(* IEC 61131-3 sources: AXOpen/src/data/ctrl/src, 20 files *)

(* ---- AxoDataCrudTask.st ---- *)
USING AXOpen.Core;

NAMESPACE AXOpen.Data

    ///<summary>
    /// Provides remote execution for CRUD operations.
    /// > [!NOTE]
    /// > This is an extension of <see cref="AxoTask"/>task see the documentatio for details about implementation in .NET.
    /// </summary>
    {#ix-set:AttributeName = "<#Data operation#>"}
    {S7.extern=ReadWrite}
    CLASS AxoDataCrudTask EXTENDS AxoRemoteTask IMPLEMENTS IAxoDataCrudTaskEntityExistState
        VAR PUBLIC
            ///<summary>
            /// Gets or sets the type of CRUD operation to be perfomed.
            /// </summary>
            CrudOperation : eCrudOperation;
            DataEntityIdentifier : STRING[254];
            _exist : BOOL;
        END_VAR

        VAR PRIVATE
            _LastCrudOperation : eCrudOperation;
            _LastDataEntityIdentifier : STRING[254];
        END_VAR
        ///<summary>
        /// Invokes this task.
        /// </summary>
        /// <param name="identifier">Data entity identifier</param>
        /// <param name="operation">Operation to perfom.</param>
        METHOD PUBLIC Invoke : IAxoTaskState
            VAR_INPUT
                identifier : STRING[254];
                operation : eCrudOperation;
            END_VAR

            // This may produce unwanted side effects if the task is invoked with different parameters while it is running.
            // It may prevent done state to be provided upstream to the caller.
            IF SUPER.IsDone() THEN
                IF (_LastDataEntityIdentifier   <> identifier OR
                    _LastCrudOperation          <> operation ) THEN
                    SUPER.Restore();
                END_IF;
            END_IF;

            IF SUPER.IsReady() THEN
                DataEntityIdentifier := identifier;
                CrudOperation := operation;
            END_IF;

            _LastDataEntityIdentifier   := DataEntityIdentifier;
            _LastCrudOperation          := CrudOperation;

            Invoke := SUPER.Invoke();
        END_METHOD

        METHOD PUBLIC Exist : BOOL
            Exist := _exist;
        END_METHOD

    END_CLASS

    TYPE
        eCrudOperation : (Create, Read, Update, Delete, CreateOrUpdate, EntityExist);
    END_TYPE
END_NAMESPACE

(* ---- AxoDataPersistentCurdTask.st ---- *)
USING AXOpen.Core;
NAMESPACE AXOpen.Data
    ///<summary>
    /// Provides remote execution for CRUD operations.
    /// > [!NOTE]
    /// > This is an extension of <see cref="AxoTask"/>task see the documentation for details about implementation in .NET.
    /// </summary>
    {#ix-set:AttributeName = "<#Data operation#>"}
    {S7.extern=ReadWrite}
    CLASS AxoDataPersistentCurdTask EXTENDS AxOpen.Core.AxoRemoteTask IMPLEMENTS  IAxoDataCrudTaskEntityExistState
        VAR PUBLIC
            ///<summary>
            /// Gets or sets the type of CRUD operation to be perfomed.
            /// </summary>
            CrudOperation : ePersistentOperation;
            DataEntityIdentifier : STRING[254];
            _exist : BOOL;
        END_VAR

        ///<summary>
        /// Invokes this task.
        /// </summary>
        /// <param name="identifier">Data entity identifier</param>
        /// <param name="operation">Operation to perfom.</param>
        METHOD PUBLIC Invoke : IAxoTaskState
            VAR_INPUT
                identifier : STRING[254];
                operation : ePersistentOperation;
            END_VAR
            CrudOperation := operation;
            DataEntityIdentifier := identifier;
            Invoke := SUPER.Invoke();
        END_METHOD

        METHOD PUBLIC Exist : BOOL
            Exist := _exist;
        END_METHOD

    END_CLASS

    TYPE
        ePersistentOperation : (Read, Update, EntityExist, UpdateAll, ReadAll);
    END_TYPE

END_NAMESPACE

(* ---- AxoDataEntityExistTask.st ---- *)
USING AXOpen.Core;

NAMESPACE AXOpen.Data
    ///<summary>
    /// Extends AxoRemoteTask for data operation within AxoData
    /// </summary>
    CLASS AxoDataEntityExistTask
        EXTENDS AxoDataExchangeTask
        IMPLEMENTS IAxoDataEntityExistTask
        VAR PUBLIC
            _exist : BOOL;
        END_VAR

        METHOD PUBLIC Exist : BOOL
            Exist := _exist;
        END_METHOD
    END_CLASS

    INTERFACE PUBLIC IAxoDataEntityExistTask EXTENDS IAxoTaskState
        METHOD Exist : BOOL END_METHOD
    END_INTERFACE

END_NAMESPACE

(* ---- AxoDataExchangeBase.st ---- *)
USING AXOpen.Core;

NAMESPACE AXOpen.Data
    ///<summary>
    /// Represents base class of data exchange.
    /// This class is used to provide abstract information about the type that can be used in rcc.
    /// </summary>
    INTERFACE PUBLIC AxoDataExchangeBase EXTENDS AXOpen.Core.IAxoObject
    END_INTERFACE
END_NAMESPACE

(* ---- IAxoDataCrudTaskEntityExistState.st ---- *)
NAMESPACE AXOpen.Data
    INTERFACE PUBLIC IAxoDataCrudTaskEntityExistState EXTENDS AXOpen.Core.IAxoTaskState
            METHOD Exist : BOOL END_METHOD
    END_INTERFACE
END_NAMESPACE

(* ---- IAxoDataEntity.st ---- *)
NAMESPACE AXOpen.Data
    INTERFACE IAxoDataEntity
        METHOD SetId
            VAR_INPUT
                Id : STRING[254];
            END_VAR
        END_METHOD
        METHOD GetId : STRING[254] END_METHOD

    END_INTERFACE
END_NAMESPACE

(* ---- IAxoDataExchange.st ---- *)
USING AXOpen.Core;

NAMESPACE AXOpen.Data
    ///<summary>
    /// Provides abastaction for data exchange.
    /// </summary>
    INTERFACE IAxoDataExchange
        METHOD Create : IAxoTaskState
            VAR_INPUT
                inIdentifier : STRING[254];
            END_VAR
        END_METHOD

        METHOD Read : IAxoTaskState
            VAR_INPUT
                inIdentifier : STRING[254];
            END_VAR
        END_METHOD

        METHOD Update : IAxoTaskState
            VAR_INPUT
                inIdentifier : STRING[254];
            END_VAR
        END_METHOD

        METHOD Delete : IAxoTaskState
            VAR_INPUT
                inIdentifier : STRING[254];
            END_VAR
        END_METHOD

        METHOD EntityExist : IAxoDataCrudTaskEntityExistState
            VAR_INPUT
                inIdentifier : STRING[254];
            END_VAR
        END_METHOD

        METHOD CreateOrUpdate : IAxoTaskState
            VAR_INPUT
                inIdentifier : STRING[254];
            END_VAR
        END_METHOD

        METHOD Restore
        END_METHOD

        METHOD Run
            VAR_INPUT
                inParent : IAxoObject;
            END_VAR
        END_METHOD
    END_INTERFACE
END_NAMESPACE

(* ---- IDataEntity.st ---- *)
NAMESPACE AXOpen.Data
    INTERFACE IDataEntity

    END_INTERFACE
END_NAMESPACE

(* ---- IDataExchange.st ---- *)
USING AXOpen.Core;

NAMESPACE ix.framework.data
    INTERFACE IDataExchange
        METHOD Create : IAxoTaskState
            VAR_INPUT
                Identifier : STRING[254];
            END_VAR
        END_METHOD

        METHOD Read : IAxoTaskState
            VAR_INPUT
                Identifier : STRING[254];
            END_VAR
        END_METHOD

        METHOD Update : IAxoTaskState
            VAR_INPUT
                Identifier : STRING[254];
            END_VAR
        END_METHOD

        METHOD Delete : IAxoTaskState
            VAR_INPUT
                Identifier : STRING[254];
            END_VAR
        END_METHOD

        METHOD Restore
        END_METHOD
    END_INTERFACE
END_NAMESPACE

(* ---- AxoDataCrudTaskEntityExistsSatisfied.st ---- *)
NAMESPACE AXOpen.Data

    ///<summary>
    /// Represents the satisfied state of a data CRUD task entity existence check.
    /// </summary>
    CLASS PUBLIC AxoDataCrudTaskEntityExistsSatisfied EXTENDS AXOpen.Core.AxoTaskStateSatisfied IMPLEMENTS IAxoDataCrudTaskEntityExistState
        VAR PRIVATE
            _exists : BOOL;
        END_VAR

        ///<summary>
        /// Returns true when the entity exists. Prior to calling this method you should call Satisfy.
        /// </summary>
        METHOD PUBLIC Exist : BOOL
            Exist := _exists;
            _exists := FALSE;
        END_METHOD

        ///<summary>
        /// Satisfies the task state by setting the existence status.
        /// </summary>
        METHOD PUBLIC Satisfy : IAxoDataCrudTaskEntityExistState
            VAR_INPUT
                inStatus : eAxoTaskState;
                inDoesExist : BOOL;
            END_VAR
            Status := inStatus;
            _exists := inDoesExist;
            Satisfy := THIS;
        END_METHOD
    END_CLASS
END_NAMESPACE

(* ---- AxoDataEntity.st ---- *)
USING AXOpen.Core;
NAMESPACE AXOpen.Data
    ///<summary>
    /// Base class for any exchangable data in <see cref="AxoDataExchange"/>.
    /// </summary>
    {S7.extern=ReadWrite}
    CLASS AxoDataEntity IMPLEMENTS IAxoDataEntity
        VAR PUBLIC
            ///<summary>
            /// Gets or sets data entity identifier.
            /// </summary>
            {#ix-attr:[RenderIgnore()]}
            DataEntityId : STRING[254];
        END_VAR

        METHOD PUBLIC SetId
            VAR_INPUT
                Id : STRING[254];
            END_VAR
            DataEntityId := Id;
        END_METHOD

        METHOD PUBLIC GetId : STRING[254]
            GetId := DataEntityId;
        END_METHOD
    END_CLASS
END_NAMESPACE

(* ---- AxoDataExchange.st ---- *)
USING AXOpen.Core;

NAMESPACE AXOpen.Data
    ///<summary>
    /// Provides base class for any data exchange with an arbitrary remote repository.
    /// </summary>
    {#ix-generic:<TOnline, TPlain>}
    {S7.extern=ReadWrite}
    CLASS AxoDataExchange EXTENDS AxoObject IMPLEMENTS IAxoDataExchange, AxoDataExchangeBase
        VAR PUBLIC
            Operation : AxoDataCrudTask;
        END_VAR

        ///<summary>
        /// Runs intialization and cyclical handling of this AxoDataExchange.
        /// </summary>
        /// <param name="parent">Parent of this object</param>
        METHOD PUBLIC OVERRIDE Run
            VAR_INPUT
                inParent : IAxoObject;
            END_VAR
            SUPER.Run(inParent);
            // Operation.Run(THIS);
            Operation.Execute(THIS);
        END_METHOD

        ///<summary>
        /// Creates new entry into the remote repository from data entity of this AxoDataExchange.
        /// </summary>
        /// <param name="identifier">Data identifier.</param>
        METHOD PUBLIC Create : IAxoTaskState
            VAR_INPUT
                identifier : STRING[254];
            END_VAR
            Create := Operation.Invoke(identifier, eCrudOperation#Create);
        END_METHOD

        ///<summary>
        /// Reads data from remote repository and copies them into data entity of this AxoDataExchange.
        /// </summary>
        /// <param name="identifier">Data identifier.</param>
        METHOD PUBLIC Read : IAxoTaskState
            VAR_INPUT
                identifier : STRING[254];
            END_VAR
            Read := Operation.Invoke(identifier, eCrudOperation#Read);
        END_METHOD

        ///<summary>
        /// Updates data in remote repository from data entiry of this AxoDataExchange.
        /// </summary>
        /// <param name="identifier">Data identifier.</param>
        METHOD PUBLIC Update : IAxoTaskState
            VAR_INPUT
                identifier : STRING[254];
            END_VAR
            Update := Operation.Invoke(identifier, eCrudOperation#Update);
        END_METHOD

        ///<summary>
        /// Deletes data entry with given ID from remote repository.
        /// </summary>
        /// <param name="identifier">Data identifier.</param>
        METHOD PUBLIC Delete : IAxoTaskState
            VAR_INPUT
                identifier : STRING[254];
            END_VAR
            Delete := Operation.Invoke(identifier, eCrudOperation#Delete);
        END_METHOD

        ///<summary>
        /// Check if data entry exists with given ID in remote repository.
        /// </summary>
        /// <param name="identifier">Data identifier.</param>
        METHOD PUBLIC EntityExist : IAxoDataCrudTaskEntityExistState
            VAR_INPUT
                identifier : STRING[254];
            END_VAR
            Operation.Invoke(identifier, eCrudOperation#EntityExist);
            EntityExist := Operation;
        END_METHOD

        ///<summary>
        /// Creates or Updates data in remote repository from data entiry of this AxoDataExchange.
        /// </summary>
        /// <param name="identifier">Data identifier.</param>
        METHOD PUBLIC CreateOrUpdate : IAxoTaskState
            VAR_INPUT
                identifier : STRING[254];
            END_VAR
            CreateOrUpdate := Operation.Invoke(identifier, eCrudOperation#CreateOrUpdate);
        END_METHOD

        ///<summary>
        /// Restores all tasks associated with this object.
        ///</summary>
        METHOD PUBLIC Restore
            Operation.Restore();
        END_METHOD
    END_CLASS
END_NAMESPACE

(* ---- AxoDataExchangeTask.st ---- *)
USING AXOpen.Core;

NAMESPACE AXOpen.Data
    ///<summary>
    /// Extends AxoRemoteTask for data operation within AxoData
    /// </summary>
    CLASS AxoDataExchangeTask
        EXTENDS AXOpen.Core.AxoRemoteTask
        VAR PUBLIC
            DataEntityIdentifier : STRING[254];
        END_VAR

        METHOD PUBLIC Invoke : IAxoTaskState
            VAR_INPUT
                identifier : STRING[254];
            END_VAR
            DataEntityIdentifier := identifier;
            Invoke := SUPER.Invoke();
        END_METHOD
    END_CLASS

END_NAMESPACE

(* ---- AxoDataFragmentExchange.st ---- *)
USING AXOpen.Core;
NAMESPACE AXOpen.Data
    ///<summary>
    /// Provides base class for any composite/fragmetes data exchange combining one or more AxoDataExchange object.
    /// </summary>
    {S7.extern=ReadWrite}
    CLASS PUBLIC AxoDataFragmentExchange EXTENDS AxoObject IMPLEMENTS IAxoDataExchange, AxoDataExchangeBase
        VAR PUBLIC
            Operation : AxoDataCrudTask;
        END_VAR

        ///<summary>
        /// Creates new entry into each associated remote repository from respective data entity.
        /// </summary>
        /// <param name="identifier">Data identifier.</param>
        METHOD PUBLIC Create : IAxoTaskState
            VAR_INPUT
                inIdentifier : STRING[254];
            END_VAR
            Create := Operation.Invoke(inIdentifier, eCrudOperation#Create);
        END_METHOD

        ///<summary>
        /// Reads data from each associated remote repository and copies it into respective data entities.
        /// </summary>
        /// <param name="identifier">Data identifier.</param>
        METHOD PUBLIC Read : IAxoTaskState
            VAR_INPUT
                inIdentifier : STRING[254];
            END_VAR
            Read := Operation.Invoke(inIdentifier, eCrudOperation#Read);
        END_METHOD

        ///<summary>
        /// Updates data in each associated remote repository from respective data entities.
        /// </summary>
        /// <param name="identifier">Data identifier.</param>
        METHOD PUBLIC Update : IAxoTaskState
            VAR_INPUT
                inIdentifier : STRING[254];
            END_VAR
            Update := Operation.Invoke(inIdentifier, eCrudOperation#Update);
        END_METHOD

        ///<summary>
        /// Deletes data entry from each associated remote repository with given ID.
        /// </summary>
        /// <param name="identifier">Data identifier.</param>
        METHOD PUBLIC Delete : IAxoTaskState
            VAR_INPUT
                inIdentifier : STRING[254];
            END_VAR
            Delete := Operation.Invoke(inIdentifier, eCrudOperation#Delete);
        END_METHOD

        ///<summary>
        /// Check if data entry exists in each associated remote repository with given ID.
        /// </summary>
        /// <param name="identifier">Data identifier.</param>
        METHOD PUBLIC EntityExist : IAxoDataCrudTaskEntityExistState
            VAR_INPUT
                inIdentifier : STRING[254];
            END_VAR
            Operation.Invoke(inIdentifier, eCrudOperation#EntityExist);
            EntityExist := Operation;
        END_METHOD

        ///<summary>
        /// Creates or Updates data entry from each associated remote repository with given ID.
        /// </summary>
        /// <param name="identifier">Data identifier.</param>
        METHOD PUBLIC CreateOrUpdate : IAxoTaskState
            VAR_INPUT
                inIdentifier : STRING[254];
            END_VAR
            CreateOrUpdate := Operation.Invoke(inIdentifier, eCrudOperation#CreateOrUpdate);
        END_METHOD

        METHOD PUBLIC Restore
            Operation.Restore();
        END_METHOD

        ///<summary>
        /// Runs intialization and cyclical handling of this AxoDataExchange.
        /// </summary>
        /// <param name="parent">Parent of this object</param>
        METHOD PUBLIC OVERRIDE Run
            VAR_INPUT
                inParent : IAxoObject;
            END_VAR
            SUPER.Run(inParent);
            // Operation.Run(THIS);
            Operation.Execute(THIS);
        END_METHOD

    END_CLASS
END_NAMESPACE

(* ---- AxoDataLocalExchange.st ---- *)
NAMESPACE AXOpen.Data
    USING AXOpen.Core;

    ///<summary>
    /// Base class for any exchangable data in <see cref="AxoDataExchange"/>.
    /// </summary>
    {S7.extern=ReadWrite}
    CLASS PUBLIC ABSTRACT AxoDataLocalExchange EXTENDS AxoObject IMPLEMENTS IAxoDataExchange
        VAR  PROTECTED
            operation : eCrudOperation;
            dataExchangeTask : AxoTask;
        END_VAR

        METHOD PUBLIC Run
            VAR_INPUT
                inParent : IAxoObject;
            END_VAR
            ;
        END_METHOD

        METHOD PUBLIC ABSTRACT Create : IAxoTaskState
            VAR_INPUT
                Identifier : STRING[254];
            END_VAR

        END_METHOD

        METHOD PUBLIC ABSTRACT Read : IAxoTaskState
            VAR_INPUT
                Identifier : STRING[254];
            END_VAR

        END_METHOD

        METHOD PUBLIC ABSTRACT Update : IAxoTaskState
            VAR_INPUT
                Identifier : STRING[254];
            END_VAR

        END_METHOD

        METHOD PUBLIC ABSTRACT Delete : IAxoTaskState
            VAR_INPUT
                Identifier : STRING[254];
            END_VAR

        END_METHOD

        METHOD PUBLIC ABSTRACT EntityExist : IAxoEntityExistTaskState
            VAR_INPUT
                Identifier : STRING[254];
            END_VAR

        END_METHOD

        METHOD PUBLIC ABSTRACT CreateOrUpdate : IAxoTaskState
            VAR_INPUT
                Identifier : STRING[254];
            END_VAR

        END_METHOD

        METHOD PUBLIC Restore
            ;
        END_METHOD
    END_CLASS
END_NAMESPACE

(* ---- AxoDataPersistentExchange.st ---- *)
USING AXOpen.Core;
NAMESPACE AXOpen.Data
    {S7.extern=ReadWrite}
    CLASS PUBLIC AxoDataPersistentExchange EXTENDS AXOpen.Core.AxoObject
        VAR PUBLIC
            Operation : AxoDataPersistentCurdTask;
        END_VAR

        VAR CONSTANT
            DEFAULT_ID : STRING := 'default';
        END_VAR

        VAR
            _IsFirstReadAllDone  : BOOL := FALSE;

            // concurrent invoke handling...
            LastCallerIdentity : ULINT;
            LastCycleCount : ULINT;
            LastOperation : ePersistentOperation;

        END_VAR

        VAR PRIVATE
            _context : IAxoContext;
        END_VAR

        ///<summary>
        /// This method determines if the current call is concurrent or not.
        ///  It takes an AXOpen.Core.IAxoObject as input and returns a BOOL.
        /// The logic involves checking the identity of the caller and comparing it with the last caller identity,
        /// along with the operation's readiness and cycle count checks.
        /// </summary>
        /// <param name="caller">IAxoObject for identifying the caller in the context of concurrent calls</param>
        METHOD PRIVATE IsNotConcurrentCall : BOOL
            VAR_INPUT
                caller : AXOpen.Core.IAxoObject;
            END_VAR
            VAR
                newCallerIdentity : ULINT;
                newCycleCount : ULINT;
                operationState : eAxoTaskState;
            END_VAR

            IsNotConcurrentCall := false;
            newCallerIdentity := caller.GetIdentity();
            newCycleCount := THIS.GetContext().OpenCycleCount();

            IF newCallerIdentity = ULINT#0 THEN // IF IDENTITY IS NOT SET DO NOT ALLOW CALL
                RETURN;
            END_IF;

            IF  newCallerIdentity = LastCallerIdentity THEN
                IsNotConcurrentCall := true;
                LastCycleCount := newCycleCount;
                RETURN;
            ELSE
                operationState := Operation.GetState();
                IF (operationState = eAxoTaskState#Ready) OR (operationState = eAxoTaskState#Done)  THEN
                    IF LastCycleCount > newCycleCount THEN // counter overflow
                        IsNotConcurrentCall := true;
                        LastCycleCount := newCycleCount;
                        LastCallerIdentity := newCallerIdentity;
                        Operation.Restore();

                    ELSIF  (LastCycleCount + ULINT#2) < newCycleCount THEN
                        IsNotConcurrentCall := true;
                        LastCycleCount := newCycleCount;
                        LastCallerIdentity := newCallerIdentity;
                        Operation.Restore();
                    END_IF;
                END_IF;
            END_IF;

        END_METHOD

        ///<summary>
        /// Runs intialization and cyclical handling of this AxoDataPersistentExchange.
        /// </summary>
        /// <param name="parent">Parent of this object</param>
        METHOD PUBLIC OVERRIDE Run
            VAR_INPUT
                inParent : IAxoObject;
            END_VAR

            IF inParent = NULL THEN
                RETURN;
            END_IF;

            IF _context = NULL THEN
                SUPER.Run(inParent);
                Operation.Run(THIS);
                _context := THIS.GetContext();
            END_IF;

            Operation.Execute(THIS);

            IF NOT _IsFirstReadAllDone THEN
                IF Operation.IsInitialized AND (Operation.Identity <> ULINT#0) THEN // MUST BE INITIALIZED AND WITH IDENTITY
                    IF Operation.IsReady() THEN // read all after startup
                        Operation.Invoke('', ePersistentOperation#ReadAll);
                        LastOperation := ePersistentOperation#ReadAll;

                    ELSIF Operation.IsDone() AND (LastOperation = ePersistentOperation#ReadAll) THEN
                         _IsFirstReadAllDone := TRUE;
                    END_IF;
                END_IF;
            END_IF;
        END_METHOD

        ///<summary>
        /// Executes the restore Operation for the AxoDataPersistentExchange component.
        /// </summary>
        METHOD PUBLIC Restore
            Operation.Restore();
        END_METHOD

        /// <summary>
        /// Return last result of EntitiyExist Operation. True = Record Exist.
        /// </summary>
        METHOD PUBLIC EntityExistResult : BOOL
            EntityExistResult := Operation._exist;
        END_METHOD

        /// <summary>
        /// This method attempts to invoke a read operation.
        /// It checks if the call is concurrent and, if not,
        /// invokes the read operation on the Operation object.
        /// </summary>
        /// <param name="caller">IAxoObject for identifying the caller in the context of concurrent calls</param>
        /// <param name="identifier">The data identifier for the persistent group.</param>
        METHOD PUBLIC InvokeRead : BOOL
            VAR_INPUT
                caller : IAxoObject;
                identifier : STRING[254];
            END_VAR

            InvokeRead := false;
            IF _IsFirstReadAllDone THEN
                IF THIS.IsNotConcurrentCall(caller) THEN
                    InvokeRead := Operation.Invoke(identifier, ePersistentOperation#Read).IsBusy();
                    LastOperation := ePersistentOperation#Read;
                END_IF;
            END_IF;
        END_METHOD

        /// <summary>
        /// This method attempts to invoke a read operation.
        /// It checks if the call is concurrent and, if not,
        /// invokes the read operation on the Operation object.
        /// </summary>
        /// <param name="caller">IAxoObject for identifying the caller in the context of concurrent calls</param>
        METHOD PUBLIC InvokeReadDefault : BOOL
            VAR_INPUT
                caller : IAxoObject;
            END_VAR
            InvokeReadDefault := false;

            IF _IsFirstReadAllDone THEN
                IF THIS.IsNotConcurrentCall(caller) THEN
                    InvokeReadDefault := Operation.Invoke(DEFAULT_ID, ePersistentOperation#Read).IsBusy();
                    LastOperation := ePersistentOperation#Read;
                END_IF;
            END_IF;
        END_METHOD

        /// <summary>
        /// This method attempts to invoke a update operation.
        /// It checks if the call is concurrent and, if not,
        /// invokes the update operation on the Operation object.
        /// </summary>
        /// <param name="caller">IAxoObject for identifying the caller in the context of concurrent calls</param>
        /// <param name="identifier">The data identifier for the persistent group.</param>
        METHOD PUBLIC InvokeUpdate : BOOL
            VAR_INPUT
                Caller : IAxoObject;
                identifier : STRING[254];
            END_VAR
            InvokeUpdate := false;

            IF _IsFirstReadAllDone THEN
                IF THIS.IsNotConcurrentCall(Caller) THEN
                    InvokeUpdate := Operation.Invoke(identifier, ePersistentOperation#Update).IsBusy();
                    LastOperation := ePersistentOperation#Update;
                END_IF;
            END_IF;
        END_METHOD

        /// <summary>
        /// This method attempts to invoke a update operation.
        /// It checks if the call is concurrent and, if not,
        /// invokes the update operation on the Operation object.
        /// </summary>
        /// <param name="caller">IAxoObject for identifying the caller in the context of concurrent calls</param>
        METHOD PUBLIC InvokeUpdateDefault : BOOL
            VAR_INPUT
                Caller : IAxoObject;
            END_VAR
            InvokeUpdateDefault := false;

            IF _IsFirstReadAllDone THEN
                IF THIS.IsNotConcurrentCall(Caller) THEN
                    InvokeUpdateDefault := Operation.Invoke(DEFAULT_ID, ePersistentOperation#Update).IsBusy();
                    LastOperation := ePersistentOperation#Update;
                END_IF;
            END_IF;
        END_METHOD

        /// <summary>
        /// This method attempts to invoke a updateAll operation.
        /// It checks if the call is concurrent and, if not,
        /// invokes the update operation on the Operation object.
        /// </summary>
        /// <param name="caller">IAxoObject for identifying the caller in the context of concurrent calls</param>
        /// <param name="identifier">The data identifier for the persistent group.</param>
        METHOD PUBLIC InvokeUpdateAll : BOOL
            VAR_INPUT
                Caller : IAxoObject;
            END_VAR
            InvokeUpdateAll := false;

            IF _IsFirstReadAllDone THEN
                IF THIS.IsNotConcurrentCall(Caller) THEN
                    InvokeUpdateAll := Operation.Invoke('', ePersistentOperation#UpdateAll).IsBusy();
                    LastOperation := ePersistentOperation#UpdateAll;
                END_IF;
            END_IF;
        END_METHOD

        /// <summary>
        /// This method attempts to invoke a readAll operation.
        /// It checks if the call is concurrent and, if not,
        /// invokes the readAll operation on the Operation object.
        /// </summary>
        /// <param name="caller">IAxoObject for identifying the caller in the context of concurrent calls</param>
        /// <param name="identifier">The data identifier for the persistent group.</param>
        METHOD PUBLIC InvokeReadAll : BOOL
            VAR_INPUT
                Caller : IAxoObject;
            END_VAR
            InvokeReadAll := false;

            IF _IsFirstReadAllDone THEN
                IF THIS.IsNotConcurrentCall(Caller) THEN
                    InvokeReadAll := Operation.Invoke('', ePersistentOperation#ReadAll).IsBusy();
                    LastOperation := ePersistentOperation#ReadAll;
                END_IF;
            END_IF;
        END_METHOD

        /// <summary>
        /// This method attempts to invoke a update operation.
        /// It checks if the call is concurrent and, if not,
        /// invokes the update operation on the Operation object.
        /// </summary>
        /// <param name="caller">IAxoObject for identifying the caller in the context of concurrent calls</param>
        /// <param name="identifier">The data identifier for the persistent group.</param>
        METHOD PUBLIC InvokeEntityExist : BOOL
            VAR_INPUT
                Caller : IAxoObject;
                identifier : STRING[254];
            END_VAR

            InvokeEntityExist := false;
            IF _IsFirstReadAllDone THEN
                IF THIS.IsNotConcurrentCall(Caller) THEN
                    InvokeEntityExist := Operation.Invoke(identifier, ePersistentOperation#EntityExist).IsBusy();
                    LastOperation := ePersistentOperation#EntityExist;
                END_IF;
            END_IF;
        END_METHOD

        /// <summary>
        /// Determines whether a read operation has been completed.
        /// </summary>
        /// <param name="caller">The object representing the caller of the method, used to check for concurrent calls.</param>
        /// <returns>Boolean indicating whether the read operation was completed.</returns>
        METHOD PUBLIC IsReadDone : BOOL
            VAR_INPUT
                caller : IAxoObject;
            END_VAR
            IsReadDone := false;

            IF _IsFirstReadAllDone THEN
                IF THIS.IsNotConcurrentCall(caller) THEN
                    IF LastOperation = ePersistentOperation#Read THEN
                        IsReadDone := Operation.IsDone();
                    END_IF;
                END_IF;
            END_IF;
        END_METHOD

        /// <summary>
        /// Determines whether a update operation has been completed.
        /// </summary>
        /// <param name="caller">The object representing the caller of the method, used to check for concurrent calls.</param>
        /// <returns>Boolean indicating whether the read operation was completed.</returns>
        METHOD PUBLIC IsUpdateDone : BOOL
            VAR_INPUT
                caller : IAxoObject;
            END_VAR
            IsUpdateDone := false;

            IF _IsFirstReadAllDone THEN
                IF THIS.IsNotConcurrentCall(caller) THEN
                    IF LastOperation = ePersistentOperation#Update THEN
                        IsUpdateDone := Operation.IsDone();
                    END_IF;
                END_IF;
            END_IF;
        END_METHOD

        /// <summary>
        /// Determines whether a updateAll operation has been completed.
        /// </summary>
        /// <param name="caller">The object representing the caller of the method, used to check for concurrent calls.</param>
        /// <returns>Boolean indicating whether the updateAll operation was completed.</returns>
        METHOD PUBLIC IsUpdateAllDone : BOOL
            VAR_INPUT
                caller : IAxoObject;
            END_VAR
            IsUpdateAllDone := false;

            IF _IsFirstReadAllDone THEN
                IF THIS.IsNotConcurrentCall(caller) THEN
                    IF LastOperation = ePersistentOperation#UpdateAll THEN
                        IsUpdateAllDone := Operation.IsDone();
                    END_IF;
                END_IF;
            END_IF;
        END_METHOD

         /// <summary>
        /// Determines whether a readAll operation has been completed.
        /// </summary>
        /// <param name="caller">The object representing the caller of the method, used to check for concurrent calls.</param>
        /// <returns>Boolean indicating whether the readAll operation was completed.</returns>
        METHOD PUBLIC IsReadAllDone : BOOL
            VAR_INPUT
                caller : IAxoObject;
            END_VAR
            IsReadAllDone := false;

            IF _IsFirstReadAllDone THEN
                IF THIS.IsNotConcurrentCall(caller) THEN
                    IF LastOperation = ePersistentOperation#ReadAll THEN
                        IsReadAllDone := Operation.IsDone();
                    END_IF;
                END_IF;
            END_IF;
        END_METHOD

        /// <summary>
        /// Determines whether a entityExist operation has been completed.
        /// </summary>
        /// <param name="caller">The object representing the caller of the method, used to check for concurrent calls.</param>
        /// <returns>Boolean indicating whether the entityExist operation was completed.</returns>
        METHOD PUBLIC IsEntityExistDone : BOOL
            VAR_INPUT
                caller : IAxoObject;
            END_VAR
            IsEntityExistDone := false;

            IF _IsFirstReadAllDone THEN
                IF THIS.IsNotConcurrentCall(caller) THEN
                    IF LastOperation = ePersistentOperation#EntityExist THEN
                        IsEntityExistDone := Operation.IsDone();
                    END_IF;
                END_IF;
            END_IF;
        END_METHOD

        /// <summary>
        /// Checks if the first read operation has been completed.
        /// </summary>
        /// <returns>Boolean indicating whether the first read operation is done.</returns>
        METHOD PUBLIC IsFirstReadDone : BOOL
            IsFirstReadDone  := _IsFirstReadAllDone;
        END_METHOD

        //!!! INTERNAL USAGE ONLY !!!
        METHOD INTERNAL SetFirstReadDone : BOOL
            _IsFirstReadAllDone  := TRUE;
        END_METHOD

    END_CLASS

END_NAMESPACE

(* ---- DataEntity.st ---- *)
NAMESPACE ix.framework.data
    CLASS DataEntity IMPLEMENTS IDataEntity
        VAR PUBLIC
            {#ix-attr:[RenderIgnore("ShadowControl", "Control")]}
            DataEntityId : STRING[254];
        END_VAR
    END_CLASS
END_NAMESPACE

(* ---- DataExchange.st ---- *)
USING ix.framework.core;

NAMESPACE ix.framework.data
    CLASS DataExchange EXTENDS IxObject
        VAR PUBLIC
           {#ix-set:AttributeName =  "<#Create#>"}
           CreateTask  : DataExchangeTask;
           {#ix-set:AttributeName =  "<#Read#>"}
           ReadTask    : DataExchangeTask;
           {#ix-set:AttributeName =  "<#Update#>"}
           UpdateTask  : DataExchangeTask;
           {#ix-set:AttributeName =  "<#Delete#>"}
           DeleteTask  : DataExchangeTask;
        END_VAR

        METHOD PUBLIC Run
            CreateTask.Initialize(THIS);
            ReadTask.Initialize(THIS);
            UpdateTask.Initialize(THIS);
            DeleteTask.Initialize(THIS);

            CreateTask.Execute();
            ReadTask.Execute();
            UpdateTask.Execute();
            DeleteTask.Execute();
        END_METHOD

        METHOD PUBLIC Create : IIxTaskState
            VAR_INPUT
                Identifier : STRING[254];
            END_VAR
            Create := CreateTask.Invoke(Identifier);
        END_METHOD

        METHOD PUBLIC Read : IIxTaskState
            VAR_INPUT
                Identifier : STRING[254];
            END_VAR
            Read := ReadTask.Invoke(Identifier);
        END_METHOD

        METHOD PUBLIC Update : IIxTaskState
            VAR_INPUT
                Identifier : STRING[254];
            END_VAR
            Update := UpdateTask.Invoke(Identifier);
        END_METHOD

        METHOD PUBLIC Delete : IIxTaskState
            VAR_INPUT
                Identifier : STRING[254];
            END_VAR
            Delete := DeleteTask.Invoke(Identifier);
        END_METHOD
    END_CLASS
END_NAMESPACE

(* ---- DataExchangeTask.st ---- *)
USING AXOpen.Core;
NAMESPACE AXOpen.Data
    CLASS DataExchangeTask EXTENDS AXOpen.Core.AxoRemoteTask
        VAR PUBLIC
            DataEntityIdentifier : STRING[254];
        END_VAR

        METHOD PUBLIC Invoke : IAxoTaskState
            VAR_INPUT
                identifier : STRING[254];
            END_VAR

            DataEntityIdentifier := identifier;
            Invoke := SUPER.Invoke();
        END_METHOD
    END_CLASS
END_NAMESPACE

(* ---- something.st ---- *)
NAMESPACE SomethingRatherThanNothig
    CLASS something
        VAR

        END_VAR

    END_CLASS
END_NAMESPACE
